// TIA Portal V17 export
// export: Created 2026-04-13T11:12:04.0578785Z, ExportSetting WithDefaults, DisplayName Totally Integrated Automation Portal, DisplayVersion V17 Update 4, DisplayName TIA Portal Openness, DisplayVersion V17 Update 4, DisplayName TIA Portal Version Control Interface, DisplayVersion V17, DisplayName SINAMICS Startdrive Advanced, DisplayVersion V17, DisplayName SINAMICS Startdrive G130, G150, S120, S150, SINAMICS MV, S210, DisplayVersion V17, DisplayName SINAMICS Startdrive G110M, G120, G120C, G120D, G120P, G115D, DisplayVersion V17, DisplayName STEP 7 Professional, DisplayVersion V17 Update 4, DisplayName STEP 7 Safety, DisplayVersion V17, DisplayName WinCC Professional, DisplayVersion V17 Update 4
FUNCTION_BLOCK "A4-脉冲控制"   // FB11, SCL
{ S7_Optimized_Access := 'TRUE' }
VERSION : 0.1
// stored: AutoNumber true, IsIECCheckEnabled false, IsRetainMemResEnabled false, MemoryReserve 100, SetENOAutomatically false, UDAEnableTagReadback false
   VAR
      主塔气锤 { S7_SetPoint := 'True'} : "A3-脉冲轮询";
      二级旋风振打锤 { S7_SetPoint := 'True'} : "A3-脉冲轮询";
      一级旋风振打锤 { S7_SetPoint := 'True'} : "A3-脉冲轮询";
      一级旋风振荡器 { S7_SetPoint := 'True'} : "A3-脉冲轮询";
      布袋气锤 { S7_SetPoint := 'True'} : "A3-脉冲轮询";
      布袋反吹 { S7_SetPoint := 'True'} : "A3-脉冲轮询";
      设备振打 { S7_SetPoint := 'True'} : "A3-脉冲轮询";
      输送出料 { S7_SetPoint := 'True'} : "A3-脉冲轮询";
      布袋出料 { S7_SetPoint := 'True'} : "A3-脉冲轮询";
      一级旋风出料 { S7_SetPoint := 'True'} : "A3-脉冲轮询";
      二级旋风出料 { S7_SetPoint := 'True'} : "A3-脉冲轮询";
      布袋出料1 { S7_SetPoint := 'True'} : "A9-循环下料控制";
      一级旋风出料1 { S7_SetPoint := 'True'} : "A9-循环下料控制";
      二级旋风出料1 { S7_SetPoint := 'True'} : "A9-循环下料控制";
      LT1 : Real := 5.0;
   END_VAR
BEGIN
   REGION 脉冲控制
       #一级旋风振打锤(num:=1,
                On_Time:=0.2,
                output_1=>"QYJ一级旋风振打锤",
                Stop_Time:="SV".YJ一级旋风振打间隔,
                脉冲开关:="MYJ一级旋风振打锤");

       #二级旋风振打锤(num := 1,
                On_Time := 0.2,
                output_1 => "QEJ二级旋风振打锤",
                Stop_Time:="SV".EJ二级旋风振打间隔,
                脉冲开关 := "MEJ二级旋风振打锤");

       #一级旋风振荡器(num := 1,
                On_Time := "SV".YJ一级旋风振荡运行,
                output_1 => "QYJ一级旋风振荡器",
                Stop_Time := "SV".YJ一级旋风振荡停止,
                脉冲开关 := "MYJ一级旋风振荡器");


       #主塔气锤(num := 4,
              On_Time := 0.2,
              output_1 => "QZT主塔气锤1",
              output_2 => "QZT主塔气锤2",
              output_3 => "QZT主塔气锤3",
              output_4 => "QZT主塔气锤4",
              Stop_Time := "SV".ZT主塔振打间隔,
              脉冲开关 := "MZT主塔气锤");

       #布袋气锤(num := 2,
              On_Time := 0.2,
              output_1 => "QCC除尘气锤1",
              output_2 => "QCC除尘气锤2",
              Stop_Time := "SV".BD布袋振打时间,
              脉冲开关 := "MCC除尘气锤");

       (* #布袋反吹(num := 2,
              On_Time := 0.2,
              output_1 => "QCC除尘气锤1",
              output_2 => "QCC除尘气锤2",
              Stop_Time := "SV".BD布袋振打时间,
              脉冲开关 := "MCC除尘气锤"); *)

        #设备振打(num := 1,
              On_Time := 0.2,
              output_1 => "QSB设备振打",
              Stop_Time := "SV".SB设备振打间隔,
              脉冲开关 := "MSB设备振打");



        (* #输送出料(num := 2,
              On_Time := 0.2,
              output_1 => "QCC除尘气锤1",
              output_2 => "QCC除尘气锤2",
              Stop_Time := "SV".BD布袋振打时间,
              脉冲开关 := "MCC除尘气锤"); *)

   (*     #布袋出料(num := 2,
              On_Time := "SV".BD布袋T出料设定,
              output_1 => "MCC除尘出料上阀",
              output_2 => "MCC除尘出料下阀",
              Stop_Time := "SV".BD布袋出料设定,
              脉冲开关 := "MBD布袋出料");

        #一级旋风出料(num := 2,
                On_Time := "SV".YJ一级旋风T出料设定,
              output_1 => "MYJ一级出料上阀",
              output_2 => "MYJ一级出料下阀",
              Stop_Time := "SV".YJ一级旋风出料设定,
              脉冲开关 := "MYJ一级出料");

      #二级旋风出料(num := 2,
              On_Time :="SV".EJ二级旋风T出料设定,
              output_1 => "MEJ二级出料上阀",
              output_2 => "MEJ二级出料下阀",
              Stop_Time :="SV".EJ二级旋风出料设定 ,
              脉冲开关 := "MEJ二级出料"); *)


        IF "PW".MS模式设定 = 1.0 OR "PW".MS模式设定 = 3.0 THEN

            #布袋出料1(下料启动开关 := "MBD布袋出料",
                   上卸料阀工作时间 := "SV".BD布袋上阀开时间,
                   上卸料阀关闭时间 := "SV".BD布袋上阀关时间,
                   下卸料阀工作时间 := "SV".BD布袋下阀开时间,
                   下卸料阀关闭时间 := "SV".BD布袋下阀关时间,
                   上下料阀 := "MCC除尘出料上阀",
                   下下料阀 := "MCC除尘出料下阀");


            #一级旋风出料1(下料启动开关 := "MYJ一级出料",
                     上卸料阀工作时间 := "SV".YJ一级旋风上阀开时间,
                     上卸料阀关闭时间 := "SV".YJ一级旋风上阀关时间,
                     下卸料阀工作时间 := "SV".YJ一级旋风下阀开时间,
                     下卸料阀关闭时间 := "SV".YJ一级旋风下阀关时间,
                     上下料阀 := "MYJ一级出料上阀",
                     下下料阀 := "MYJ一级出料下阀");

            #二级旋风出料1(下料启动开关 := "MEJ二级出料",
                     上卸料阀工作时间 := "SV".EJ二级旋风上阀开时间,
                     上卸料阀关闭时间 := "SV".EJ二级旋风上阀关时间,
                     下卸料阀工作时间 := "SV".EJ二级旋风下阀开时间,
                     下卸料阀关闭时间 := "SV".EJ二级旋风下阀关时间,
                     上下料阀 := "MEJ二级出料上阀",
                     下下料阀 := "MEJ二级出料下阀");

        END_IF;


   END_REGION
END_FUNCTION_BLOCK
